FUNCTION_BLOCK FB_TcLogger EXTENDS FB_AbstractLogger
VAR
END_VAR

// https://github.com/PeterZerlauth/Tc3_Component

METHOD M_Log
VAR_INPUT
	stEvent	: 		ST_Event;
END_VAR

VAR
	sMessage:			STRING(255);
END_VAR
IF stEvent.eEventType >= eLogLevel THEN
	sMessage:= Concat(Concat(stEvent.sInstance, ' | '), stEvent.sDefault);
	CASE stEvent.eEventType OF
		E_Event.Error:
			ADSLOGSTR( msgCtrlMask := ADSLOG_MSGTYPE_ERROR , msgFmtStr := '%s', strArg := sMessage);
		E_Event.Warning:
			ADSLOGSTR( msgCtrlMask := ADSLOG_MSGTYPE_WARN , msgFmtStr := '%s', strArg := sMessage);
		E_Event.Information:
			ADSLOGSTR( msgCtrlMask := ADSLOG_MSGTYPE_HINT , msgFmtStr := '%s', strArg := sMessage);
		E_Event.Debug:
			ADSLOGSTR( msgCtrlMask := ADSLOG_MSGTYPE_HINT, msgFmtStr := '%s', strArg := sMessage);
		E_Event.Verbose:
			ADSLOGSTR( msgCtrlMask := ADSLOG_MSGTYPE_HINT , msgFmtStr := '%s', strArg := sMessage);
	END_CASE
END_IF
END_METHOD

END_FUNCTION_BLOCK

(* stored: Version 1.1.0.1
   POU FB_TcLogger: Id {bea54b82-5a5b-4b7e-85c1-9b16a6ed125e}, SpecialFunc None
   Method M_Log: Id {9de4bedf-a79b-482f-8aed-4ec654fd7e05} *)
